FUNCTION_BLOCK A_1State_10Transitions (* Basic FB with empty ECC *)
  (* Standard: 61499-2 *)
  (* Version 1.0, 2023-09-22, AK124910 *)
  PACKAGE servSeq;
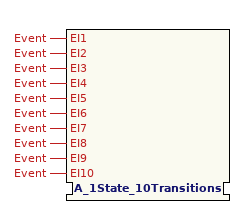
  EVENT_INPUT
    EI1;
    EI2;
    EI3;
    EI4;
    EI5;
    EI6;
    EI7;
    EI8;
    EI9;
    EI10;
  END_EVENT
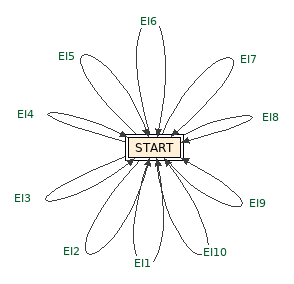
  EC_STATES
    START; (* Initial State *)
  END_STATES
  EC_TRANSITIONS
    START TO START := EI1;
    START TO START := EI2;
    START TO START := EI3;
    START TO START := EI4;
    START TO START := EI5;
    START TO START := EI6;
    START TO START := EI7;
    START TO START := EI8;
    START TO START := EI9;
    START TO START := EI10;
  END_TRANSITIONS
  (* Service external/internal_interface: Basic FB with empty ECC *)
END_FUNCTION_BLOCK
